# EPICS substitutions: nsls2emApp/Db/StatusDoubleReg.substitutions
file db/StatusDoubleReg.template
{pattern
{RegOffset-Double,Reg}
{0,Reg0}
{8,Reg1}
{16,Reg2}
{24,Reg3}
}
